(* PLC project sample_project, sample_company sample_product 1 *)
(* stored: creationDateTime 2024-07-18T21:30:47, modificationDateTime 2024-07-18T22:03:54 *)

FUNCTION_BLOCK sample_function_block_FBD
  VAR
    T1 : TON;  (* The temperature is decreased on a time delay, when the comepressor has been activated *)
    P_Cooling : TIME := TIME#500ms;
    xReduceTemp : BOOL;  (* Signal for dereasing the temperature *)
    T2 : TON;  (* The temperature is increased on a time delay, when the compressor has been activated *)
    P_Environment : TIME := TIME#2s0ms;  (* Delay time when the door is closed *)
    P_EnvironmentDoorOpen : TIME := TIME#1s0ms;  (* Delay time when the door is open *)
    xRaiseTemp : BOOL;  (* Signal for increasing the temperature *)
    timTemp : TIME;  (* Delay time *)
    iCounter : STATISTICS_INT := (IN := (IN := 5, RESET := TRUE, MN := 100, MX := -100, AVG := 1, SUM := 2, COUNTER := 3), RESET := TRUE, MN := 100, MX := -100, AVG := 1, SUM := 2, COUNTER := 3);
    newVar1 : ARRAY[0..5] OF ARRAY[0..5] OF R_TRIG := [[(CLK := TRUE, Q := TRUE), 4(()), (CLK := TRUE, Q := TRUE)], 3([6(())]), [3(()), (CLK := TRUE, Q := TRUE), 2(())], [6(())]];
    newVar : ARRAY[0..5] OF F_TRIG := [(CLK := TRUE, Q := TRUE), 3(()), (CLK := TRUE, Q := TRUE), ()];
  END_VAR
  VAR  (* added by the conversion: wires and edge detectors of the diagram *)
    _SEL4_OUT : ANY;
  END_VAR

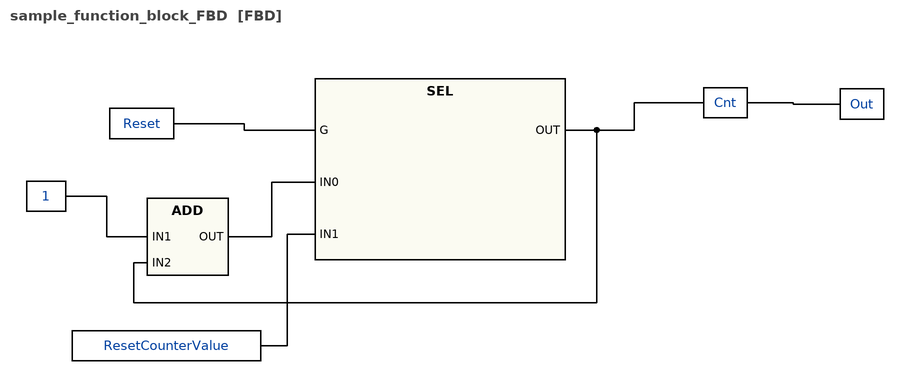
(* FBD diagram, written out as Structured Text *)
Out := Cnt;
_SEL4_OUT := SEL(Reset, 1 + _SEL4_OUT, ResetCounterValue);
Cnt := _SEL4_OUT;
END_FUNCTION_BLOCK

(* Counter in ST language *)
FUNCTION_BLOCK sample_function_block_ST
  VAR_INPUT
    Reset : BOOL;
  END_VAR
  VAR_OUTPUT
    Out : INT;
  END_VAR
  VAR
    Cnt : INT;
  END_VAR
  VAR_EXTERNAL CONSTANT
    ResetCounterValue : INT;
  END_VAR

      IF Reset THEN
  Cnt := ResetCounterValue;
ELSE
  Cnt := Cnt + 1;
END_IF;

Out := Cnt;
     
END_FUNCTION_BLOCK

PROGRAM sample_program
  VAR_INPUT
    Reset : BOOL := TRUE;
  END_VAR
  VAR_OUTPUT
    Cnt0 : INT := 1;
    Cnt1 : INT := 2;
    Cnt2 : INT := 3;
    Cnt3 : INT := 4;
    Cnt4 : INT := 5;
  END_VAR
  VAR
    sample_function_block_ST0 : sample_function_block_ST;
    sample_function_block_FBD0 : sample_function_block_FBD;
  END_VAR

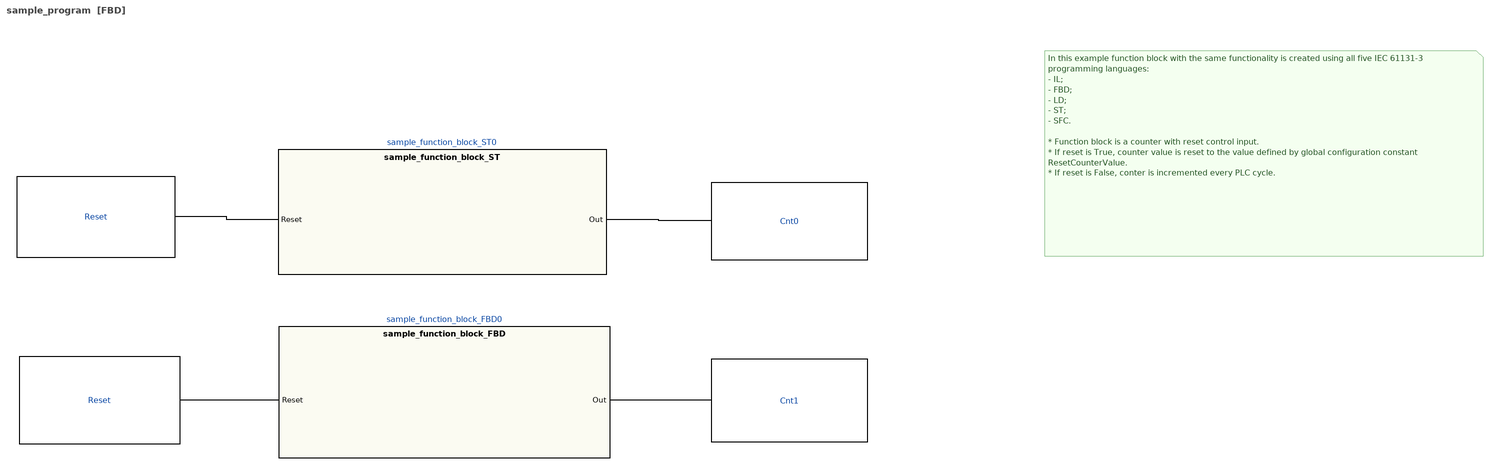
(* FBD diagram, written out as Structured Text *)
(* In this example function block with the same functionality is created using all five IEC 61131-3 programming languages:
- IL;
- FBD;
- LD;
- ST;
- SFC.

* Function block is a counter with reset control input.
* If reset is True, counter value is reset to the value defined by global configuration constant ResetCounterValue.
* If reset is False, conter is incremented every PLC cycle. *)
sample_function_block_ST0(Reset := Reset);
Cnt0 := sample_function_block_ST0.Out;
sample_function_block_FBD0(Reset := Reset);
Cnt1 := sample_function_block_FBD0.Out;
END_PROGRAM

CONFIGURATION sample_config
  VAR_GLOBAL CONSTANT
    ResetCounterValue : INT := 17;
  END_VAR
  RESOURCE sample_resource ON PLC
    TASK sample_task(INTERVAL := T#200ms, PRIORITY := 0);
    PROGRAM sample_task_instance WITH sample_task : sample_program;
  END_RESOURCE
END_CONFIGURATION
